FUNCTION_BLOCK FB_ADD
VAR_INPUT
	in1,in2,in3:INT;
END_VAR
VAR_OUTPUT
	out:INT;
END_VAR
VAR
END_VAR

out:=in1+in2+in3;

END_FUNCTION_BLOCK

(* stored: Version 1.1.0.1, ProductVersion 3.1.4024.12
   POU FB_ADD: Id {45864090-ed79-4cb7-a422-594959bc984a}, SpecialFunc None *)
